TYPE ST_ergonomic_data :
STRUCT
	head_height:REAL;
	head_angle:REAL;
	arm_height:REAL;
	foot_distance:REAL;
END_STRUCT
END_TYPE

(* stored: Version 1.1.0.1, ProductVersion 3.1.4024.11
   DUT ST_ergonomic_data: Id {476619f7-fa03-4b2e-ad16-ef2a94d0f41f} *)
